TYPE EcSoeRead_CMD_typ :
	STRUCT
		Enable	: BOOL ;
	END_STRUCT
END_TYPE

(* stored: Version 1.1.0.1, ProductVersion 3.1.4024.3
   DUT EcSoeRead_CMD_typ: Id {aead690c-a497-0654-0149-f4f5b41c3e49} *)
